// Mitsubishi GX Works2 project: 19   PLC: FX3G

// task Task_01 (event TRUE, interval 0, priority 31): POU_01

PROGRAM POU_01
VAR
  wstep : INT;
  ton1 : TON;
END_VAR
M99 := FALSE AND
M0 AND M1 AND M2 AND M3 AND M4 AND 
M5 AND M6 AND M7 AND 
Y0 AND Y1 AND Y2;

IF M8002 THEN
    wstep := 0;
END_IF;

IF M0 THEN
    wstep := 100;
END_IF;

CASE wstep OF
    0:
        TON1(in := FALSE);
        
        IF (M1) THEN
            wstep := wstep + 1;
        END_IF;
    1:
        Y0 := TRUE;

        IF M3 THEN
            wstep := 20;
        END_IF;
        IF M2 THEN
            wstep := 40;
        END_IF;

    20:
        IF M4 THEN
            wstep := wstep + 1;
        END_IF;
    21:
        Y0 := FALSE;
        Y1 := TRUE;
        TON1(in := NOT TON1.Q, pt := T#5s);

        IF (TON1.Q) THEN
            wstep := wstep + 1;
        END_IF;
    22:
        Y0 := TRUE;
        Y1 := FALSE;

        IF (M5) THEN
            wstep := wstep + 1;
        END_IF;
    23:
        Y0 := FALSE;
        Y2 := TRUE;
        TON1(in := NOT TON1.Q, pt := T#15s);

        IF (TON1.Q) THEN
            wstep := wstep + 1;
        END_IF;
    24:
        Y0 := TRUE;
        Y2 := FALSE;

        IF (M6) THEN
            wstep := wstep + 1;
        END_IF;
    25:
        Y0 := FALSE;
        TON1(in := TRUE, pt := T#20s);

        IF (TON1.Q AND M7) THEN
            wstep := 0;
        END_IF;

    40:
        IF M6 THEN
            wstep := 41;
        END_IF;
    41:
        Y0 := FALSE;
        TON1(in := TRUE, pt := T#20s);
        
        IF (TON1.Q AND M7) THEN
            wstep := 0;
        END_IF;

    100:
        ZRST(TRUE, Y0, Y2);

        IF NOT M0 THEN
            wstep := 0;
        END_IF;
END_CASE;
END_PROGRAM
